// LS Electric XG5000 project: 테스트
// PLC LSPLC

PROGRAM NewProgram (task: 스캔 프로그램)

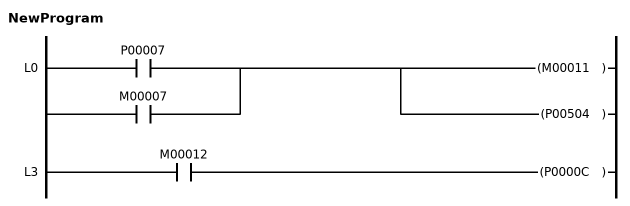
; L0
LOAD      P00007
OR        M00007
OUT       M00011
OUT       P00504
; L3
LOAD      M00012
OUT       P0000C